(* IEC 61131-3 sources: UserLog/, 2 files *)

(* ---- UserLog.fun ---- *)
FUNCTION UserLogBasic : UDINT (*Write to the User logbook synchronously*)
	VAR_INPUT
		Severity : DINT; (*Use UserLogSeverityEnum or arEVENTLOG_SEVERITY constants*)
		Code : UINT; (*0..65535*)
		Message : STRING[0]; (*Event description*)
	END_VAR
END_FUNCTION

FUNCTION UserLogAdvanced : UDINT (*Write to the User logbook with runtime data*)
	VAR_INPUT
		Severity : DINT; (*Use UserLogSeverityEnum or arEVENTLOG_SEVERITY constants*)
		Code : UINT; (*0..65535*)
		Message : STRING[0]; (*Event description with optional format specifiers*)
		Values : UserLogFormatType; (*Format values to replace specifiers (%b, %f, %i, %s)*)
	END_VAR
END_FUNCTION

FUNCTION UserLogCustom : UDINT (*Write to any user logbook synchronously*)
	VAR_INPUT
		Logbook : STRING[0]; (*Name of logbook*)
		Severity : DINT; (*Use UserLogSeverityEnum or arEVENTLOG_SEVERITY constants*)
		Facility : UINT; (*0..4095*)
		Code : UINT; (*0..65535*)
		Origin : ArEventLogRecordIDType; (*(Optional) Origin record ID*)
		Object : STRING[0]; (*(Optional) Object name*)
		Message : STRING[0]; (*Event description with optional format specifiers*)
		Values : UserLogFormatType; (*Format values to replace specifiers (%b, %f, %i, %s)*)
	END_VAR
END_FUNCTION

FUNCTION UserLogEventText : UDINT (*Write to any user logbook through binary-encoded data and event texts*)
	VAR_INPUT
		Logbook : STRING[0]; (*Name of logbook*)
		Event : DINT; (*Event ID (match Text ID)*)
		Origin : ArEventLogRecordIDType; (*(Optional) Origin record ID*)
		Object : STRING[0]; (*(Optional) Object name*)
		Message : STRING[0]; (*Ordedred list of specifiers (%b, %i, %f, %s) to replace the placeholders in the event text ({1}, {2}, ...)*)
		Values : UserLogFormatType; (*Format values to replace specifiers (%b, %f, %i, %s)*)
	END_VAR
END_FUNCTION

FUNCTION UserLogCreate : DINT (*Create a custom logbook in an Init subroutine*)
	VAR_INPUT
		Name : STRING[0]; (*Name of logbook limited to 10 characters*)
		Size : UDINT; (*Size of logbook in bytes (minimum 4096)*)
	END_VAR
END_FUNCTION

FUNCTION UserLogSetSeverityLevel : DINT (*Suppress messages below the input level and return previous level*)
	VAR_INPUT
		Level : DINT; (*Severity level threshold*)
	END_VAR
END_FUNCTION

FUNCTION UserLogGetSeverity : USINT (*Get ArEventLog severity from an event ID*)
	VAR_INPUT
		Event : DINT; (*Event ID*)
	END_VAR
END_FUNCTION

FUNCTION UserLogGetFacility : UINT (*Get ArEventLog facility from an event ID*)
	VAR_INPUT
		Event : DINT; (*Event ID*)
	END_VAR
END_FUNCTION

FUNCTION UserLogGetCode : UINT (*Get ArEventLog code from an event ID*)
	VAR_INPUT
		Event : DINT; (*Event ID*)
	END_VAR
END_FUNCTION

(* ---- UserLog.var ---- *)
VAR CONSTANT
	USERLOG_MESSAGE_LENGTH : UDINT := 120; (*Maximum length of all messages written to user logbooks*)
	USERLOG_FACILITY : UINT := 10; (*Facility number used for UserLogBasic and UserLogAdvanced functions*)
	USERLOG_ERROR_IDENT : DINT := -515234032; (*An error occurred when calling ArEventLogGetIdent. See User logbook for details*)
	USERLOG_ERROR_WRITE : DINT := -515234022; (*An error occurred when calling ArEventLogWrite. See User logbook for details*)
	USERLOG_ERROR_CREATE : DINT := -515234012; (*An error occurred when calling ArEventLogCreate. See User logbook for details*)
	USERLOG_FORMAT_INDEX : USINT := 5; (*Maximum index of each runtime data type*)
	USERLOG_FORMAT_LENGTH : USINT := 80; (*Length of string runtime data*)
	USERLOG_EXAMPLE_TEXT_ID : DINT := 1611615776; (*Example Text ID (Event ID) for UserLogEventText function*)
END_VAR
